Omron Sysmac Studio project RingBufferExample_FallbackLogger (Sysmac Studio 1.62.0.9, StandardProject)
(* Examples for RingBufferLib. *)

# Controller Example: NX102-9000 version 1.64
Task Main (priority 4, period or condition 2000): PseudoMain, ProgramLoader
Task Subsystem (priority 18, period or condition 10000): LogFileWriter, LogSender, RedundantLogSender
Library FileStreamWriterLib 0.0.1 (contents left out)
Library ModeManagerLib 0.0.2 (contents left out)
Library UdpClientLib 0.0.1 (contents left out)
Library RingBufferLib 0.0.2 (contents left out)
Library FileStreamReaderLib 0.0.2 (contents left out)
Library TcpClientLib 0.0.1 (contents left out)

TYPE RetainedRingBufferContext : STRUCT
    Context : stfreakjp\buf\RingBufferContext;
    InitialContext : stfreakjp\buf\RingBufferContext;
    Inited : BOOL;
END_STRUCT END_TYPE

VAR_GLOBAL RETAIN
    gpLoggerBufferContext : RetainedRingBufferContext;
    gpLoggerBuffer : ARRAY[0..32767] OF BYTE;
END_VAR

PROGRAM README
RETURN;
(*

# About This Project
This project demonstrates the RingBufferLib.
It showcases logging by combining RingBufferLib with FileStreamWriterLib, FileStreamReaderLib, and TcpClientLib.
This allows for simultaneous writing of logs to the controller's SD card and sending them to a remote TCP endpoint.

Furthermore, if sending to the TCP endpoint fails, it **falls back** to writing to the SD card.
When the TCP endpoint connection is restored,
the logs that were output during the fallback period are then sent to a dedicated TCP endpoint for fallback logs.

The logger uses its buffer as holding memory to retain values even after a power loss.
Additionally, when writing logs to the SD card or sending them to a remote TCP endpoint,
the output programs also refer to logs the logger wrote before those programs started.

# About the Programs
This project includes the following programs:

* POU/Program/ProgramLoader
    Selects the program to execute.

* POU/Program/PseudoMain
    Continuously generates logs.

* POU/Program/LogFileWriter
    Outputs logs to the controller's SD card.

* POU/Program/LogSender
    Sends logs to a remote TCP endpoint.

* POU/Program/RedundantLogSender
    Sends logs to redundant remote UDP endpoints.

* POU/Program/SimpleTcpMonitor_ps1
    A PowerShell script to set up a TCP endpoint.

* POU/Program/SimpleUdpMonitor_ps1
    A PowerShell script to set up a UDP endpoint.

* POU/Program/StartMultiTcpMonitors_ps1
    A PowerShell script to launch four TCP endpoints in Windows Terminal.

# Usage Steps
Use this program by following these steps:

1.  Configure the project for your environment.
    Match the controller model and ensure access to the network you're using.

2.  Adjust `POU/Program/LogUdpSender` for your environment.
    Change the values of the `REMOTE_ADDR` and `REMOTE_PORT` variables to the remote UDP endpoint that will receive the logs.
	If you're using `POU/Program/RedundantLogUdpSender`, make sure to modify that as well.

3.  Listen for TCP on an appropriate device.
    You can find a reference PowerShell script in `POU/Program/SimpleTcpMonitor_ps1`.
	`StartMultiTcpMonitors_ps1` is a PowerShell script that uses Windows Terminal to launch four TCP endpoints.

4.  Run the program on the controller.   
    Transfer the program to the controller and start its execution.

5.  Confirm that data is being sent to the opened TCP socket.

6.  Confirm that log files are created on the controller's SD card.


# このプロジェクトについて
このプロジェクトは、RingBufferLibの例示です。
RingBufferLibを使用した、FileStreamWriterLib、FileStreamReaderLibとTcpClientLibを組み合わせたロギングをデモします。
ログのコントローラのSDカードへの書き込みとリモートTCPエンドポイントへの送信を同時に行います。
また、TCPエンドポイントへの送信ができないとき、SDカード出力へフォールバックし、
TCPエンドポイントへの送信が復旧すると、フォールバックしたログをフォールバック専用のTCPエンドポイントに送信します。

ロガーは、バッファを保持メモリとして電源断を越えて値を保持します。
また、ログのSDカードへの書き込みとリモートTCPエンドポイントへの送信は、
それら出力プログラムが起動する以前にロガーが書き込んだログも参照して出力します。

# プログラムについて
このプロジェクトは、以下のプログラムを含みます。

* POU/プログラム/ProgramLoader
  実行するプログラムを選択します。

* POU/プログラム/PseudoMain
  ログを生成し続けます。

* POU/プログラム/LogFileWriter
  コントローラのSDカードにログを出力します。

* POU/プログラム/LogSender
  リモートTCPエンドポイントにログを送信します。

* POU/プログラム/RedundantLogSender
  冗長のリモートUDPエンドポイントにログを送信します。

* POU/プログラム/SimpleTcpMonitor_ps1
  TCPエンドポイントを立ち上げるPowerShellスクリプトです。

* POU/プログラム/SimpleUdpMonitor_ps1
  UDPエンドポイントを立ち上げるPowerShellスクリプトです。

* POU/プログラム/StartMultiTcpMonitors_ps1
  Windows Terminalで4つのTCPエンドポイントを立ち上げるPowerShellスクリプトです。

# 使用手順
このプログラムは、以下の手順で使用します。

1.  プロジェクトの構成を使用環境に合わせる
    コントローラの型式を合わせ、使用するネットワークにアクセスできるようにします。
  
2.  `POU/プログラム/LogSender`を使用環境に合わせる
    `REMOTE_ADDR`と`REMOTE_PORT`変数の値をログを受信するリモートTCPエンドポイントに変更します。
	`POU/プログラム/RedundantLogSender`を使用する場合、そちらも変更します。
  
3.  適当な端末でTCPをリッスンする
    `POU/プログラム/SimpleTcpMonitor_ps1`に参考のPowerShellスクリプトがあります。
	`StartMultiTcpMonitors_ps1`は、Windows Terminalを使用して4つのTCPエンドポイントを立ち上げるPowerShellスクリプトです。

4.  コントローラでプログラムを動作させる
    プログラムをコントローラに転送して動作させます。
  
5.  待ち受けているTCPソケットにデータが送られてくることを確認する

6.  コントローラのSDカードにログファイルが作成されていることを確認する


For the parts to which I have rights, I follow POU/Program/LICENSE.
You are free to use and modify it, but we are not responsible for any damage or loss related to it.

(c) 2025 KITA Munemitsu

*)
END_PROGRAM

PROGRAM ProgramLoader
VAR
    iModeManager : ModeManagerContext;
    RUN_MODE : STRING[128];
END_VAR
(*

# About This Program
This program is the selector for the execution program.
Specify the operation mode with "RUN_MODE" in "Configuration".


# このプログラムについて
このプログラムは、実行プログラムのセレクタです。
"Configuration"の"RUN_MODE"で動作モードを指定します。


(c) 2025 KITA Munemitsu

*)

// Configuration
IF P_First_Run THEN
	// "run:standalone", "run" or "run:redundant".
	RUN_MODE := 'run';
END_IF;

IF P_First_Run THEN
	ModeManager_init(Context:=iModeManager,
					 Name:='ProgramLoader',
					 OnSuccessStop:=TRUE,
					 OnFailStop:=FALSE,
					 OnFailAlarm:=TRUE,
					 AlarmCode:=1);

	ModeSet(Context:=iModeManager);
		// Logs are output to the controller's SD card.
		Mode(Context:=iModeManager, Name:='run:standalone');
			ModeUnit(Context:=iModeManager, Name:='PseudoMain');
			ModeUnit(Context:=iModeManager, Name:='LogFileWriter');

		// It outputs logs to the controller's SD card and to a remote TCP endpoint.
		Mode(Context:=iModeManager, Name:='run');
			ModeUnit(Context:=iModeManager, Name:='PseudoMain');
			ModeUnit(Context:=iModeManager, Name:='LogFileWriter');
			ModeUnit(Context:=iModeManager, Name:='LogSender');

		// It outputs logs to the controller's SD card and to two remote TCP endpoints.
		Mode(Context:=iModeManager, Name:='run:redundant');
			ModeUnit(Context:=iModeManager, Name:='PseudoMain');
			ModeUnit(Context:=iModeManager, Name:='LogFileWriter');
			ModeUnit(Context:=iModeManager, Name:='LogSender');
			ModeUnit(Context:=iModeManager, Name:='RedundantLogSender');
	ModeSetClose(Context:=iModeManager);
	
	ModeManager_selectMode(Context:=iModeManager, Name:=RUN_MODE);
END_IF;

ModeManager_activate(Context:=iModeManager);
END_PROGRAM

PROGRAM PseudoMain
VAR
    LOGGING_INTERVAL : UINT;
END_VAR
VAR RETAIN
    iCounter : ULINT := 0;
END_VAR
VAR
    iMsg : STRING[1024];
    iWaitTick : UINT;
END_VAR
VAR RETAIN
    iForceClear : BOOL;
END_VAR
VAR_EXTERNAL
    gpLoggerBuffer : ARRAY[0..32767] OF BYTE;
    gpLoggerBufferContext : RetainedRingBufferContext;
END_VAR
(*

# About This Program
This program will keep writing logs.
Setting `iForceClear` to "TRUE" will force initialization.


# このプログラムについて
このプログラムは、ログを書き続けます。
`iForceClear`を"TRUE"にすることで、強制的に初期化します。


(c) 2025 KITA Munemitsu

*)

// Configuration
IF P_First_Run THEN
	LOGGING_INTERVAL := 1;
	// iForceClear := FALSE;
END_IF;

IF P_First_Run THEN
	// Setup Logger.
	RetainedLogger_init(Context:=gpLoggerBufferContext,
						Buffer:=gpLoggerBuffer,
						ForceClear:=iForceClear);
	IF iForceClear THEN
		iCounter := 0;
		iForceClear := FALSE;
	END_IF;
	
	iMsg := CONCAT('{"boot":true',
				   CONCAT(',"lastcount":', ULINT_TO_STRING(iCounter)),
				   CONCAT(',"timestamp":"', DtToString(GetTime()), '"'),
				   '}$L');
	RetainedLogger_write(Context:=gpLoggerBufferContext,
						 Buffer:=gpLoggerBuffer,
						 Message:=iMsg);
	
	iWaitTick := LOGGING_INTERVAL;
END_IF;

// Logging at regular intervals.
Dec(iWaitTick);
IF iWaitTick < 1 THEN
	Inc(iCounter);
	iMsg := CONCAT('{"counter":', ULINT_TO_STRING(iCounter),
				   ',"timestamp":"', DtToString(GetTime()),
				   '"}$L');
	RetainedLogger_write(Context:=gpLoggerBufferContext,
						 Buffer:=gpLoggerBuffer,
						 Message:=iMsg);
	
	iWaitTick := LOGGING_INTERVAL;
END_IF;
END_PROGRAM

PROGRAM LogFileWriter
VAR
    LOG_PATH : STRING[64];
    iLogFileWriter : stfreakjp\fileio\FileStreamWriter;
    iLogFileWriterContext : stfreakjp\fileio\FileStreamWriterContext;
    iLogFileWriterBufferContext : stfreakjp\buf\RingBufferContext;
    iLogFileWriterBuffer : ARRAY[0..65534] OF BYTE;
END_VAR
VAR RETAIN
    ipLoggerWrittenTracker : stfreakjp\buf\RingBufferContext;
END_VAR
VAR_EXTERNAL
    gpLoggerBuffer : ARRAY[0..32767] OF BYTE;
    gpLoggerBufferContext : RetainedRingBufferContext;
END_VAR
(*

# About This Program
This program keeps track of the logger's buffer writes and outputs them to a file.


# このプログラムについて
このプログラムは、ロガーのバッファ書き込みを追跡してファイルに出力し続けます。


(c) 2025 KITA Munemitsu

*)

// Configuration
IF P_First_Run THEN
	LOG_PATH := '/log.txt';
END_IF;

IF P_First_Run THEN
	// Setup Log writer.
	RingBuffer_init(Context:=iLogFileWriterBufferContext,
					Buffer:=iLogFileWriterBuffer);	
	FileStreamWriter_configure(Context:=iLogFileWriterContext,
							   Activate:=TRUE,
							   Path:=LOG_PATH,
							   FileOpenMode:=_eFOPEN_MODE#_WRITE_APPEND,
							   FlushThreshold:=(SizeOfAry(iLogFileWriterBuffer) / 2),
							   FlushOnDeactivate:=TRUE);
	iLogFileWriter.Enable := TRUE;
	
	// Tracks Logger writes.
	RetainedRingBuffer_createWriteTracker(
		Target:=gpLoggerBufferContext,
		Tracker:=ipLoggerWrittenTracker);
END_IF;

// Gets the difference of the logger buffer into the log writer's write buffer.
RetainedRingBuffer_pullWrite(Context:=iLogFileWriterBufferContext,
							 Buffer:=iLogFileWriterBuffer,
							 Tracker:=ipLoggerWrittenTracker,
							 Tracked:=gpLoggerBufferContext,
							 TrackedBuffer:=gpLoggerBuffer);
iLogFileWriter(Context:=iLogFileWriterContext,
			   BufferContext:=iLogFileWriterBufferContext,
			   Buffer:=iLogFileWriterBuffer);
END_PROGRAM

PROGRAM LogSender
VAR CONSTANT
    LOG_SENDER_RESET_PAYLOAD : STRING[8] := '$$R$$L$$R$$L';
END_VAR
VAR
    FALLBACK_FILE_PATH : STRING[64];
    REMOTE_ADDR : STRING[256];
    REMOTE_PORT : UINT;
    REMOTE_FALLBACK_PORT : UINT;
    WAIT_TICKS_UNTILE_STABLE : UINT;
END_VAR
VAR CONSTANT
    STATE_REMOTE_ACTIVE : UINT := 0;
    STATE_REMOTE_INACTIVE : UINT := 1;
    STATE_FALLBACK_WAIT : UINT := 10;
    STATE_FALLBACK_HALT : UINT := 5;
    STATE_FALLBACK_ACTIVE : UINT := 20;
    STATE_FALLBACK_SENDER_ERROR : UINT := 900;
    STATE_FALLBACK_SENDER_INACTIVE : UINT := 0;
    STATE_FALLBACK_SENDER_HALT : UINT := 5;
    STATE_FALLBACK_SENDER_ACTIVE : UINT := 20;
END_VAR
VAR
    iLogSenderClient : stfreakjp\net\TcpSendClient;
    iLogSenderContext : stfreakjp\net\TcpClientContext;
END_VAR
VAR RETAIN
    iLogSenderBufferContext : stfreakjp\buf\RingBufferContext;
    iLogSenderBuffer : ARRAY[0..65534] OF BYTE;
    ipLoggerWrittenTracker : stfreakjp\buf\RingBufferContext;
END_VAR
VAR
    iFallbackLogWriter : stfreakjp\fileio\FileStreamWriter;
    iFallbackLogWriterContext : stfreakjp\fileio\FileStreamWriterContext;
END_VAR
VAR RETAIN
    iFallbackLogBufferContext : stfreakjp\buf\RingBufferContext;
    iFallbackLogBuffer : ARRAY[0..32767] OF BYTE;
END_VAR
VAR
    iFallbackLogReader : stfreakjp\fileio\FileStreamReader;
    iFallbackLogReaderContext : stfreakjp\fileio\FileStreamReaderContext;
    iFallbackLogReaderBufferContext : stfreakjp\buf\RingBufferContext;
    iFallbackLogReaderBuffer : ARRAY[0..8191] OF BYTE;
    iFallbackLogSenderContext : stfreakjp\net\TcpClientContext;
    iFallbackLogSender : stfreakjp\net\TcpSendClient;
    iState : UINT := 0;
    iStateFallback : UINT := 0;
    iStateFallbackSender : UINT := 0;
    iWaitTick : UINT;
    iFileOpenMode : _eFOPEN_MODE;
    iErrorID : WORD;
END_VAR
VAR_EXTERNAL
    gpLoggerBufferContext : RetainedRingBufferContext;
    gpLoggerBuffer : ARRAY[0..32767] OF BYTE;
END_VAR
(*

# About This Program
This program continuously **tracks logger buffer writes and sends them to a remote TCP endpoint.
If sending to the TCP endpoint isn't possible, it falls back to outputting to an SD card.
Once the TCP endpoint connection is restored,
the logs written to the SD card are then sent to a dedicated remote TCP endpoint for fallback logs.

Before running it, you must change the "REMOTE_ADDR" in "Configuration" to adjust your environment.

## Regarding Failures During Fallback
Failures can occur even while in fallback mode.
Here's how they impact the system.

*   Power Loss During Fallback Output
    Since the fallback buffer is retained, the system will output the file upon power-up.
 
*   Writer Error During Fallback Output
    Data loss is expected as autonomous recovery isn't feasible.
	The fallback functionality will cease operation.
	
*   Buffer Overflow Before Fallback Output Starts
    This will result in data loss.

*   Fallback Occurs While Sending Fallback Logs
    The system will **append new output to the existing file.
	
*   Power Loss During Fallback Transmission
    All data will be **re-sent upon power-up**.

*   Reader Error During Fallback Transmission
    If the file doesn't exist, there will be data loss.
	Fallback transmission will stop.

*   Sender Error During Fallback Transmission
    Retries will occur as long as the main sender is operational.
	If the main sender is down, fallback transmission will stop.


# このプログラムについて
このプログラムは、ロガーのバッファ書き込みを追跡してリモートのTCPエンドポイントに送信し続けます。
また、TCPエンドポイントへの送信ができないときはフォールバックしてSDカードに出力します。
そして、TCPエンドポイントへの送信が可能になるとSDカードに書き出したログを、
フォールバックを専用に受信するリモートのTCPエンドポイントに送信します。
実行前に"Configuration"の"REMOTE_ADDR"を使用環境に合わせる必要があります。

## フォールバック中の障害について
フォールバック中にも障害が発生する可能性があります。
フォールバック中の障害の影響は、以下です。

*   フォールバック出力中に電源断
    フォールバックバッファが保持なので電源入時にファイル出力。

*   フォールバック出力中にWriterがエラー
    自律的な回復が見込めないのでデータ喪失。
    フォールバック機能停止。

*   フォールバック出力開始までにバッファがオーバーフロー
    データ喪失。

*   フォールバック送信中にフォールバック発生
    ファイルに追記で出力。
  
*   フォールバック送信中に電源断
    電源入時に全て再送信。

*   フォールバック送信中にReaderがエラー
    ファイルが存在しなければデータ喪失。
    フォールバック送信停止。
  
*   フォールバック送信中にSenderがエラー
    主Senderが落ちない限り再試行。
    主Senderが落ちているときフォールバック送信停止。


(c) 2025 KITA Munemitsu

*)

// Configuration.
IF P_First_Run THEN
	REMOTE_ADDR := 'YOUR_REMOTE_DEVICE';
	REMOTE_PORT := 12101;
	REMOTE_FALLBACK_PORT := 12102;
	FALLBACK_FILE_PATH := '/log_fallback.txt';
	WAIT_TICKS_UNTILE_STABLE := 1000;
END_IF;

IF P_First_Run THEN	
	// Setup Log sender.
	//
	// The log sender monitors the logger buffer and sends the written logs.
	IF NOT RingBuffer_isInitialized(Context:=iLogSenderBufferContext) THEN
		RingBuffer_init(Context:=iLogSenderBufferContext,
						Buffer:=iLogSenderBuffer);
	END_IF;
	TcpClient_configure(Context:=iLogSenderContext,
						Activate:=TRUE,
						Destination:=REMOTE_ADDR,
						DestinationPort:=REMOTE_PORT,
						Port:=0,
						UseSend:=TRUE,
						ConnectRetryTimes:=360,
						ConnectRetryInterval:=50,
						ConnectTimeout:=10);
	iLogSenderClient.Enable := TRUE;
	
	// Tracks logger writes.
	RetainedRingBuffer_createWriteTracker(Target:=gpLoggerBufferContext,
										  Tracker:=ipLoggerWrittenTracker);

	// Sends the log sender reset payload first.
	RingBuffer_writeString(Context:=iLogSenderBufferContext,
						   Buffer:=iLogSenderBuffer,
						   Value:=LOG_SENDER_RESET_PAYLOAD);
END_IF;

// Log sender task.
CASE iState OF
	// STATE_REMOTE_ACTIVE
	0:		
		IF TcpClient_isReconnecting(Context:=iLogSenderContext) THEN
			RingBuffer_transferFully(Source:=iLogSenderBufferContext,
									 SourceBuffer:=iLogSenderBuffer,
									 Destination:=iFallbackLogBufferContext,
									 DestinationBuffer:=iFallbackLogBuffer);
			
			iState := STATE_REMOTE_INACTIVE;
		ELSE
			RetainedRingBuffer_pullWrite(Context:=iLogSenderBufferContext,
										 Buffer:=iLogSenderBuffer,
										 Tracker:=ipLoggerWrittenTracker,
										 Tracked:=gpLoggerBufferContext,
										 TrackedBuffer:=gpLoggerBuffer);
		END_IF;
		
	// STATE_REMOTE_INACTIVE
	1:	
		IF TcpClient_isActive(Context:=iLogSenderContext) THEN			
			iState := STATE_REMOTE_ACTIVE;
		ELSE
			RetainedRingBuffer_pullWrite(Context:=iFallbackLogBufferContext,
										 Buffer:=iFallbackLogBuffer,
										 Tracker:=ipLoggerWrittenTracker,
										 Tracked:=gpLoggerBufferContext,
										 TrackedBuffer:=gpLoggerBuffer);
			IF NOT TcpClient_isReconnecting(Context:=iLogSenderContext) THEN
				Inc(iState);
			END_IF;
		END_IF;

	// STATE_DOWN
	2:
		RetainedRingBuffer_pullWrite(Context:=iFallbackLogBufferContext,
									 Buffer:=iFallbackLogBuffer,
									 Tracker:=ipLoggerWrittenTracker,
									 Tracked:=gpLoggerBufferContext,
									 TrackedBuffer:=gpLoggerBuffer);			
END_CASE;
iLogSenderClient(Context:=iLogSenderContext,
				 SendBufferContext:=iLogSenderBufferContext,
				 SendBuffer:=iLogSenderBuffer);

// Fallback file writer task.
CASE iStateFallback OF
	// STATE_FALLBACK_INIT
	0:
		IF RingBuffer_isReadable(Context:=iFallbackLogBufferContext) THEN
			iStateFallback := STATE_FALLBACK_ACTIVE;
		ELSE
			RingBuffer_init(Context:=iFallbackLogBufferContext,
							Buffer:=iFallbackLogBuffer);
			
			iStateFallback := STATE_FALLBACK_WAIT;
		END_IF;
	
	// STATE_FALLBACK_HALT
	// 5:
		
	// STATE_FALLBACK_WAIT
	10:
		CASE iState OF
			// STATE_INACTIVE
			1: iStateFallback := STATE_FALLBACK_ACTIVE;
		END_CASE;
	
	// STATE_FALLBACK_ACTIVE
	20:
		CASE iStateFallbackSender OF
			// STATE_FALLBACK_SENDER_INACTIVE
			0: iFileOpenMode := _eFOPEN_MODE#_WRITE_CREATE;
		ELSE
			iFileOpenMode := _eFOPEN_MODE#_WRITE_APPEND;
		END_CASE;
		FileStreamWriter_configure(Context:=iFallbackLogWriterContext,
								   Activate:=TRUE,
								   Path:=FALLBACK_FILE_PATH,
								   FileOpenMode:=iFileOpenMode,
								   FlushThreshold:=(SizeOfAry(iFallbackLogBuffer) / 2),
								   FlushOnDeactivate:=TRUE);
		iFallbackLogWriter.Enable := TRUE;
		
		Inc(iStateFallback);
	21:
		CASE iState OF
			// STATE_REMOTE_ACTIVE
			0:
				FileStreamWriter_deactivate(Context:=iFallbackLogWriterContext);
				iFallbackLogWriter.Enable := FALSE;

				Inc(iStateFallback);
		ELSE			
			IF FileStreamWriter_hasError(Context:=iFallbackLogWriterContext) THEN
				FileStreamWriter_deactivate(Context:=iFallbackLogWriterContext);
				iFallbackLogWriter.Enable := FALSE;
				
				iStateFallback := STATE_FALLBACK_HALT;
			ELSE
				RetainedRingBuffer_pullWrite(Context:=iFallbackLogBufferContext,
											 Buffer:=iFallbackLogBuffer,
											 Tracker:=ipLoggerWrittenTracker,
											 Tracked:=gpLoggerBufferContext,
											 TrackedBuffer:=gpLoggerBuffer);	
			END_IF;
		END_CASE;
	22:
		IF NOT iFallbackLogWriter.Busy THEN
			IF FileStreamWriter_hasError(COntext:=iFallbackLogWriterContext) THEN
				iStateFallback := STATE_FALLBACK_HALT;
			ELSE	
				iWaitTick := MAX(UINT#1, WAIT_TICKS_UNTILE_STABLE);
			
				Inc(iStateFallback);
			END_IF;
		END_IF;
	23:
		Dec(iWaitTick);
		CASE iState OF
			// STATE_REMOTE_INACTIVE
			1:
				FileStreamWriter_configure(Context:=iFallbackLogWriterContext,
										   Activate:=TRUE,
										   Path:=FALLBACK_FILE_PATH,
										   FileOpenMode:=_eFOPEN_MODE#_WRITE_APPEND,
										   FlushThreshold:=(SizeOfAry(iFallbackLogBuffer) / 2),
										   FlushOnDeactivate:=TRUE);
				iFallbackLogWriter.Enable := TRUE;

				iStateFallback := iStateFallback - 2;
		ELSE
			IF iWaitTick < 1 THEN
				CASE iStateFallbackSender OF
					// STATE_FALLBACK_SENDER_INACTIVE
					0: iStateFallbackSender := STATE_FALLBACK_SENDER_ACTIVE;
				END_CASE;
				
				iStateFallback := STATE_FALLBACK_WAIT;
			END_IF;
		END_CASE;
END_CASE;
iFallbackLogWriter(Context:=iFallbackLogWriterContext,
				   BufferContext:=iFallbackLogBufferContext,
				   Buffer:=iFallbackLogBuffer);

// Fallbacked log sender task.
CASE iStateFallbackSender OF
	// STATE_FALLBACK_SENDER_INACTIVE
	// 0:
	
	// STATE_FALLBACK_SENDER_HALT
	// 5:
	
	// STATE_FALLBACK_SENDER_ACTIVE
	20:
		RingBuffer_init(Context:=iFallbackLogReaderBufferContext,
						Buffer:=iFallbackLogReaderBuffer);
		TcpClient_configure(Context:=iFallbackLogSenderContext,
							Activate:=TRUE,
							Destination:=REMOTE_ADDR,
							DestinationPort:=REMOTE_FALLBACK_PORT,
							Port:=0,
							UseSend:=TRUE,
							ConnectRetryTimes:=20,
							ConnectRetryInterval:=100,
							ConnectTimeout:=100);
		iFallbackLogSender.Enable := TRUE;
		FileStreamReader_configure(Context:=iFallbackLogReaderContext,
								   Activate:=TRUE,
								   Path:=FALLBACK_FILE_PATH,
								   ReadThreshold:=(SizeOfAry(iFallbackLogReaderBuffer) / 2));
		iFallbackLogReader.Enable := TRUE;
		
		Inc(iStateFallbackSender);
	21:
		IF TcpClient_hasError(Context:=iFallbackLogSenderContext) THEN
			iStateFallbackSender := iStateFallbackSender + 6;
		ELSIF TcpClient_isActive(Context:=iFallbackLogSenderContext) THEN
			FileStreamReader_activate(Context:=iFallbackLogReaderContext);
			
			Inc(iStateFallbackSender);
		END_IF;
	22:
		IF TcpClient_hasError(Context:=iFallbackLogSenderContext)
			OR FileStreamReader_hasError(Context:=iFallbackLogReaderContext)
		THEN
			iStateFallbackSender := iStateFallbackSender + 5;
		ELSIF FileStreamReader_isEOF(Context:=iFallbackLogReaderContext) THEN			
			Inc(iStateFallbackSender);
		END_IF;
	23:
		IF TcpClient_hasError(Context:=iFallbackLogSenderContext) THEN
			iStateFallbackSender := iStateFallbackSender + 4;
		ELSIF NOT RingBuffer_isReadable(Context:=iFallbackLogReaderBufferContext) THEN
			iStateFallbackSender := iStateFallbackSender + 4;
		END_IF;
	27:
		TcpClient_deactivate(Context:=iFallbackLogSenderContext);
		FileStreamReader_deactivate(Context:=iFallbackLogReaderContext);
		iFallbackLogSender.Enable := FALSE;
		iFallbackLogReader.Enable := FALSE;
		
		Inc(iStateFallbackSender);
	28:
		IF NOT (iFallbackLogReader.Busy OR iFallbackLogReader.Busy) THEN
			Inc(iStateFallbackSender);
		END_IF;
	29:
		IF TcpClient_hasError(Context:=iFallbackLogSenderContext)
			OR FileStreamReader_getError(Context:=iFallbackLogReaderContext, ErrorID=>iErrorID)
		THEN
			CASE WORD_TO_UINT(iErrorID) OF
				16#0000, // None.
				16#1405, // Accessing file.
				16#140B: // Exceeding maximum number of open files.
					iStateFallbackSender := STATE_FALLBACK_SENDER_ERROR;
			ELSE
				iStateFallbackSender := STATE_FALLBACK_SENDER_HALT;
			END_CASE;
		ELSE
			iStateFallbackSender := STATE_FALLBACK_SENDER_INACTIVE;
		END_IF;
	
	// STATE_FALLBACK_SENDER_ERROR
	900:
		CASE iState OF
			// STATE_ACTIVE
			0: iStateFallbackSender := STATE_FALLBACK_SENDER_ACTIVE;
			// STATE_DOWN
			2: iStateFallbackSender := STATE_FALLBACK_SENDER_HALT;
		END_CASE;
END_CASE;
iFallbackLogReader(Context:=iFallbackLogReaderContext,
				   BufferContext:=iFallbackLogReaderBufferContext,
				   Buffer:=iFallbackLogReaderBuffer);
iFallbackLogSender(Context:=iFallbackLogSenderContext,
				   SendBufferContext:=iFallbackLogReaderBufferContext,
				   SendBuffer:=iFallbackLogReaderBuffer);
END_PROGRAM

PROGRAM RedundantLogSender
VAR CONSTANT
    LOG_SENDER_RESET_PAYLOAD : STRING[8] := '$$R$$L$$R$$L';
END_VAR
VAR
    REMOTE_ADDR : STRING[256];
    REMOTE_PORT : UINT;
    SENDER_PORT : UINT;
    iLogSenderUdpClient : stfreakjp\net\UdpSendClient;
    iLogSenderContext : stfreakjp\net\UdpClientContext;
    iLogSenderSendBufferContext : stfreakjp\buf\RingBufferContext;
    iLogSenderSendBuffer : ARRAY[0..8191] OF BYTE;
END_VAR
VAR RETAIN
    ipLoggerWrittenTracker : stfreakjp\buf\RingBufferContext;
END_VAR
VAR_EXTERNAL
    gpLoggerBufferContext : RetainedRingBufferContext;
    gpLoggerBuffer : ARRAY[0..32767] OF BYTE;
END_VAR
(*

# About This Program
This program acts as a redundancy for log transmission.
Before running it, you must change the "REMOTE_ADDR" in "Configuration" to adjust your environment.


# このプログラムについて
このプログラムは、ログ送信の冗長機能として動作します。
実行前に"Configuration"の"REMOTE_ADDR"を使用環境に合わせる必要があります。


(c) 2025 KITA Munemitsu

*)

// Configuration.
IF P_First_Run THEN
	REMOTE_ADDR := 'YOUR_REMOTE_DEVICE';
	REMOTE_PORT := 12002;
	SENDER_PORT := 12002;
END_IF;

IF P_First_Run THEN	
	// Setup Log sender.
	//
	// The log sender monitors the logger buffer and sends the written logs.
	//
	RingBuffer_init(Context:=iLogSenderSendBufferContext,
					Buffer:=iLogSenderSendBuffer);
	UdpClient_configure(Context:=iLogSenderContext,
						Activate:=TRUE,
						Destination:=REMOTE_ADDR,
						DestinationPort:=REMOTE_PORT,
						Port:=SENDER_PORT,
						UseSend:=TRUE);
	iLogSenderUdpClient.Enable := TRUE;
	
	// Tracks logger writes.
	RetainedRingBuffer_createWriteTracker(
		Target:=gpLoggerBufferContext,
		Tracker:=ipLoggerWrittenTracker);

	// Sends the log sender reset payload first.
	RingBuffer_writeString(Context:=iLogSenderSendBufferContext,
						   Buffer:=iLogSenderSendBuffer,
						   Value:=LOG_SENDER_RESET_PAYLOAD);
END_IF;

// Gets the difference of the logger buffer into the log sender's sending buffer.
RetainedRingBuffer_pullWrite(Context:=iLogSenderSendBufferContext,
							 Buffer:=iLogSenderSendBuffer,
							 Tracker:=ipLoggerWrittenTracker,
							 Tracked:=gpLoggerBufferContext,
							 TrackedBuffer:=gpLoggerBuffer);
iLogSenderUdpClient(Context:=iLogSenderContext,
					SendBufferContext:=iLogSenderSendBufferContext,
					SendBuffer:=iLogSenderSendBuffer);
END_PROGRAM

PROGRAM SimpleTcpMonitor_ps1
RETURN;
(*

Below is a PowerShell script that opens and listens on a TCP socket.


以下は、TCPソケットをオープンして待ち受けるPowerShellスクリプトです。

```powershell:simple-tcp-monitor.ps1
param(
    [Parameter(Mandatory=$false, Position=0)][int]$Port = 12101,
    [Parameter(Mandatory=$false, Position=0)][int]$ReadInterval = 50,
    [Parameter(Mandatory=$false, Position=1)][string]$Mode = 'jsonl'
)

function Mode-Jsonl {
    param(
        [int]$Port,
        [int]$ReadInterval
    )
    $listenerEndPoint = New-Object IPEndpoint([System.Net.IPAddress]::Any, $Port)
    $tcpListener = New-Object System.Net.Sockets.TCPListener($listenerEndpoint)
    $client = $null
    $clientStream = $null
    $reader = $null
    $task = $null
    $entity = $null
    $prevEntity = $null

    try {
        $tcpListener.Start()
        while ($true) {
            # Wait for client connection.
            if ($null -eq $client) {
                if ($null -eq $task) {
                    $task = $tcpListener.AccepttcpClientAsync()
                }
                if (-not $task.Wait(200)) {
                    continue
                }

                $client = $task.GetAwaiter().GetResult();
                $clientStream = $client.GetStream()
                $reader = New-Object System.IO.StreamReader($clientStream)
                $task = $null
            }
            if ($reader.EndOfStream) {
                $reader.Close()
                $clientStream.Close()
                $client.Close()
                $task = $null
                $reader = $null
                $clientStream = $null
                $client = $null
                $entity = $null
                $prevEntity = $null
                continue
            }

            # Waiting to receive data.
            try {
                if ($null -eq $task) {
                    $task = $reader.ReadLineAsync()
                }

                if (-not $task.Wait($ReadInterval)) {
                    continue
                }
                $entity = $task.GetAwaiter().GetResult();
                $task = $null
            }
            catch {
                Write-Host "error: $($_.Exception.Message)"
                $reader.Close()
                $clientStream.Close()
                $client.Close()
                $reader = $null
                $ClientStream = $null
                $client = $null
            }

            if ($null -ne $entity) {
                if ("" -eq $entity) {
                    if ("" -eq $prevEntity) {
                        Write-Host 'reset'
                    }
                } else {
                    try {
                        $entity | ConvertFrom-Json | Write-Host
                    }
                    catch {
                        Write-Host "error payload: ${entity}"
                    }
                }
            }

            $prevEntity = $entity
            $entity = $null
        }
    }
    catch {
        Write-Host "error: $($_.Exception.Message)"
    }
    finally {
        if ($client) {
            $reader.Close()
            $clientStream.Close()
            $client.Close()
        }
        $tcpListener.Stop()
    }
}

function Mode-Raw {
    param(
        [string]$Port,
        [int]$ReadInterval
    )
    $listenerEndPoint = New-Object IPEndpoint([System.Net.IPAddress]::Any, $Port)
    $tcpListener = New-Object System.Net.Sockets.TCPListener($listenerEndpoint)
    $client = $null
    $clientStream = $null
    $reader = $null
    $task = $null
    $prevEntity = $null

    try {
        $tcpListener.Start()
        while ($true) {
            # Wait for client connection.
            if ($null -eq $client) {
                if ($null -eq $task) {
                    $task = $tcpListener.AcceptTcpClientAsync()
                }
                if (-not $task.Wait(200)) {
                    continue
                }

                $client = $task.GetAwaiter().GetResult();
                $clientStream = $client.GetStream()
                $reader = New-Object System.IO.StreamReader($clientStream)
                $task = $null
            }
            if ($reader.EndOfStream) {
                $reader.Close()
                $clientStream.Close()
                $client.Close()
                $task = $null
                $reader = $null
                $clientStream = $null
                $client = $null
                $entity = $null
                $prevEntity = $null
                continue
            }

            # Waiting to receive data.
            try {
                if ($null -eq $task) {
                    $task = $reader.ReadLineAsync()
                }

                if (-not $task.Wait($ReadInterval)) {
                    continue
                }
                $entity = $task.GetAwaiter().GetResult();
                $task = $null
            }
            catch {
                Write-Host "error: $($_.Exception.Message)"
                $reader.Close()
                $clientStream.Close()
                $client.Close()
                $reader = $null
                $ClientStream = $null
                $client = $null
            }

            if ($null -ne $entity) {
                if ("" -eq $entity) {
                    if ("" -eq $prevEntity) {
                        Write-Host 'reset'
                    }
                } else {
                    $entity | Write-Host
                }
            }

            $prevEntity = $entity
            $entity = $null
        }
    }
    catch {
        Write-Host "error: $($_.Exception.Message)"
    }
    finally {
        if ($client) {
            $reader.Close()
            $clientStream.Close()
            $client.Close()
        }
        $tcpListener.Stop()
    }
}

switch ( $Mode )
{
    Jsonl { Mode-Jsonl -Port $Port -ReadInterval $ReadInterval }
    Raw   { Mode-Raw -Port $Port -ReadInterval $ReadInterval }
}
```
*)
END_PROGRAM

PROGRAM SimpleUdpMonitor_ps1
RETURN;
(*

Below is a PowerShell script that opens and listens on a UDP socket.


以下は、UDPソケットをオープンして待ち受けるPowerShellスクリプトです。

```powershell:simple-udp-monitor.ps1
param(
    [Parameter(Mandatory=$false, Position=0)][int]$Port = 12001,
    [Parameter(Mandatory=$false, Position=1)][string]$Mode = 'raw'
)

function Mode-Jsonl {
    param(
        [string]$Port
    )

    $udpClient = New-Object System.Net.Sockets.UdpClient($Port)
    try {
        $task = $null
        $RESET_PAYLOAD = "`r`n`r`n"
        $ENTITY_DELIMITER = "`n"
        $ENTITY_MAX_LENGTH = 8192
        $recv = $null
        $payload = $null
        $restPaylod = $null
        $entities = $null
        while ($true) {
            if ($null -eq $task) {
                $task = $udpClient.ReceiveAsync()
            }
            if (-not $task.Wait(20)) {
                continue
            }
            $receiveBytes = $task.GetAwaiter().GetResult();

            $recv = [Text.Encoding]::UTF8.GetString($receiveBytes.Buffer)
            $payload = $recv -split $RESET_PAYLOAD
            if ($payload.length -gt 1) {
                Write-Host 'reset'
                $restPaylod = ""
            }
            $entities = ($restPaylod + $payload[-1]) -split $ENTITY_DELIMITER
                | Where-Object {($_ -ne "") -and ($_.Length -le $ENTITY_MAX_LENGTH)}
            $restPaylod = ""
            foreach ($entity in $entities) {
                try {
                    $entity | ConvertFrom-Json | Write-Host
                }
                catch {
                    if ($entity -eq $entities[-1]) {
                        $restPaylod = $entity
                    }
                }
            }

            $task = $null
        }
    }
    catch {
        Write-Host "error: $($_.Exception.Message)"
    }
    finally {
        $udpClient.Close()
    }
}

function Mode-Raw {
    param(
        [string]$Port
    )

    $udpClient = New-Object System.Net.Sockets.UdpClient($Port)
    try {
        $task = $null
        $message = ''
        while ($true) {
            if ($null -eq $task) {
                $task = $udpClient.ReceiveAsync()
            }
            if (-not $task.Wait(20)) {
                continue
            }
            $receiveBytes = $task.GetAwaiter().GetResult();
            $message = [Text.Encoding]::UTF8.GetString($receiveBytes.Buffer)
            Write-Host $message -NoNewline

            $task = $null
        }
    }
    catch {
        Write-Host "error: $($_.Exception.Message)"
    }
    finally {
        $udpClient.Close()
    }
}

switch ( $Mode ) {
	Jsonl { Mode-Jsonl -Port $Port }
    Raw   { Mode-Raw -Port $Port }
}
```
*)
END_PROGRAM

PROGRAM StartMultiTcpMonitors_ps1
RETURN;
(*

Below is a PowerShell script that launches four "simple-tcp-monitor.ps" files in Windows Terminal.
Run this script while "simple-tcp-monitor.ps1" is in the same folder.


以下は、Windows Terminalで4つの"simple-tcp-monitor.ps"を立ち上げるPowerShellスクリプトです。
"simple-tcp-monitor.ps1"が同じフォルダにある状態で実行します。

```powershell:start-multi-tcp-monitors.ps1
param(
    [Parameter(Mandatory=$false, Position=0)][int[]]$Ports = @(12101, 12102, 13101, 13102),
    [Parameter(Mandatory=$false, Position=1)][string]$Mode = 'jsonl'
)

$scriptFile = "simple-tcp-monitor.ps1"
$scriptDir = Split-Path -Parent $MyInvocation.MyCommand.Definition
$scriptPath = Join-Path $scriptDir $scriptFile
if (-not (Test-Path $scriptPath)) {
    Write-Error "error: Not fount '${scriptFile}' in '${scriptPath}'"
    exit 1
}

$wtCommandString = "pwsh.exe -NoExit -Command ""&{ & `"${scriptPath}`" -Port $($Ports[0]) -Mode `"${Mode}`" }"" ; " + `
                   "split-pane -H pwsh.exe -NoExit -Command ""&{ & `"${scriptPath}`" -Port $($Ports[1]) -Mode `"${Mode}`" }"" ; " + `
                   "split-pane -V pwsh.exe -NoExit -Command ""&{ & `"${scriptPath}`" -Port $($Ports[2]) -Mode `"${Mode}`" }"" ; " + `
                   "split-pane -H pwsh.exe -NoExit -Command ""&{ & `"${scriptPath}`" -Port $($Ports[3]) -Mode `"${Mode}`" }"""

# For debug.
# Write-Host "command: wt.exe $wtCommandString"

Start-Process -FilePath "wt.exe" -ArgumentList $wtCommandString
```
*)
END_PROGRAM

PROGRAM LICENSE
RETURN;
(*
The MIT License (MIT)

Copyright(c) 2025 KITA Munemitsu

Permission is hereby granted, free of charge, to any person obtaining a copy of this software and associated
documentation files (the “Software”), to deal in the Software without restriction, including without limitation
the rights to use, copy, modify, merge, publish, distribute, sublicense, and/or sell copies of the Software,
and to permit persons to whom the Software is furnished to do so, subject to the following conditions:

The above copyright notice and this permission notice shall be included in all copies or substantial portions of the Software.

THE SOFTWARE IS PROVIDED “AS IS”, WITHOUT WARRANTY OF ANY KIND, EXPRESS OR IMPLIED, INCLUDING BUT NOT
LIMITED TO THE WARRANTIES OF MERCHANTABILITY, FITNESS FOR A PARTICULAR PURPOSE AND NONINFRINGEMENT.
IN NO EVENT SHALL THE AUTHORS OR COPYRIGHT HOLDERS BE LIABLE FOR ANY CLAIM, DAMAGES OR OTHER LIABILITY,
WHETHER IN AN ACTION OF CONTRACT, TORT OR OTHERWISE, ARISING FROM, OUT OF OR IN CONNECTION WITH THE SOFTWARE
OR THE USE OR OTHER DEALINGS IN THE SOFTWARE.
*)
END_PROGRAM

FUNCTION RetainedLogger_init : BOOL
VAR_IN_OUT
    Context : RetainedRingBufferContext;
    Buffer : ARRAY[*] OF BYTE;
END_VAR
VAR_INPUT
    ForceClear : BOOL := False;
END_VAR
IF NOT EN THEN
	RetainedLogger_init := FALSE;
	
	RETURN;
END_IF;

RetainedLogger_init
	:= RetainedRingBuffer_init(Context:=Context,
							   Buffer:=Buffer,
							   Force:=ForceClear);
END_FUNCTION

FUNCTION RetainedLogger_write : BOOL
VAR
    iBinMsg : ARRAY[0..4095] OF BYTE;
    iBinMsgSize : UINT;
END_VAR
VAR_IN_OUT
    Context : RetainedRingBufferContext;
    Buffer : ARRAY[*] OF BYTE;
END_VAR
VAR_INPUT
    Message : STRING[1986] := '';
END_VAR
IF NOT EN THEN
	RetainedLogger_write := FALSE;
	
	RETURN;
END_IF;

iBinMsgSize
	:= StringToAry(In:=Message, AryOut:=iBinMsg[0]);
RetainedLogger_write
	:= \\stfreakjp\buf\RingBuffer_write(
						   Context:=Context.Context,
						   Buffer:=Buffer,
						   In:=iBinMsg,
						   Head:=0,
						   Size:=iBinMsgSize,
						   AllowOverWrite:=TRUE);
END_FUNCTION

FUNCTION RetainedRingBuffer_init : BOOL
VAR_IN_OUT
    Context : RetainedRingBufferContext;
    Buffer : ARRAY[*] OF BYTE;
END_VAR
VAR_INPUT
    Force : BOOL := False;
END_VAR
(*

Initializes the RetainedRingBufferContext.


RetainedRingBufferContextを初期化する。


(c) 2025 KITA Munemitsu

*)

IF NOT EN THEN
	RetainedRingBuffer_init := FALSE;
	
	RETURN;
END_IF;

IF NOT Context.Inited OR Force THEN
	\\stfreakjp\buf\RingBuffer_init(
						Context:=Context.Context,
						Buffer:=Buffer);
	Context.Inited := TRUE;
END_IF;

Context.InitialContext := Context.Context;

RetainedRingBuffer_init := TRUE;
END_FUNCTION

FUNCTION RetainedRingBuffer_createWriteTracker : BOOL
VAR_IN_OUT
    Target : RetainedRingBufferContext;
END_VAR
VAR_INPUT
    UseInitial : BOOL := True;
    Force : BOOL := False;
END_VAR
VAR_IN_OUT
    Tracker : stfreakjp\buf\RingBufferContext;
END_VAR
(*

Creates a tracking context for tracking writes to the RetainedRingBuffer.


RetainedRingBufferの書き込みを追跡するための追跡コンテクストを作成する。


(c) 2025 KITA Munemitsu

*)

IF NOT EN
	OR NOT Target.Inited
THEN	
	RetainedRingBuffer_createWriteTracker := FALSE;
	
	RETURN;
END_IF;

// NOTE: Maybe we need a method to determine the validity of a tracker.
IF Target.Context.WriteSize >= Tracker.WriteSize
	AND Tracker.WriteSize <> 0
	AND NOT Force
THEN
	RetainedRingBuffer_createWriteTracker := TRUE;
	
	RETURN;
END_IF;

IF UseInitial THEN
	RetainedRingBuffer_createWriteTracker
		:= \\stfreakjp\buf\RingBuffer_createWriteTracker(
							   Target:=Target.InitialContext,
							   Tracker=>Tracker);
ELSE
	RetainedRingBuffer_createWriteTracker
		:= \\stfreakjp\buf\RingBuffer_createWriteTracker(
							   Target:=Target.Context,
							   Tracker=>Tracker);
END_IF;
END_FUNCTION

FUNCTION RetainedRingBuffer_createReadTracker : BOOL
VAR_IN_OUT
    Target : RetainedRingBufferContext;
END_VAR
VAR_INPUT
    UseInitial : BOOL := True;
    Force : BOOL := False;
END_VAR
VAR_OUTPUT
    Tracker : stfreakjp\buf\RingBufferContext;
END_VAR
(*

Creates a tracking context to track reads of the RetainedRingBuffer.


RetainedRingBufferの読み出しを追跡するための追跡コンテクストを作成する。


(c) 2025 KITA Munemitsu

*)

IF NOT EN
	OR NOT Target.Inited
THEN	
	RetainedRingBuffer_createReadTracker := FALSE;
	
	RETURN;
END_IF;

// NOTE: Maybe we need a method to determine the validity of a tracker.
IF Target.Context.ReadSize >= Tracker.ReadSize
	AND Tracker.ReadSize <> 0
	AND NOT Force
THEN
	RetainedRingBuffer_createReadTracker := TRUE;
	
	RETURN;
END_IF;

IF UseInitial THEN
	RetainedRingBuffer_createReadTracker
		:= \\stfreakjp\buf\RingBuffer_createReadTracker(
							   Target:=Target.InitialContext,
							   Tracker=>Tracker);
ELSE
	RetainedRingBuffer_createReadTracker
		:= \\stfreakjp\buf\RingBuffer_createReadTracker(
							   Target:=Target.Context,
							   Tracker=>Tracker);
END_IF;
END_FUNCTION

FUNCTION RetainedRingBuffer_createTracker : BOOL
VAR_IN_OUT
    Target : RetainedRingBufferContext;
END_VAR
VAR_INPUT
    UseInitial : BOOL := True;
    Force : BOOL := False;
END_VAR
VAR_OUTPUT
    Tracker : stfreakjp\buf\RingBufferContext;
END_VAR
(*

Creates a tracking context for tracking reads and writes to the RetainedRingBuffer.


RetainedRingBufferの読み書きを追跡するための追跡コンテクストを作成する。


(c) 2025 KITA Munemitsu

*)

IF NOT EN THEN	
	RetainedRingBuffer_createTracker := FALSE;
	
	RETURN;
END_IF;

// NOTE: Maybe we need a method to determine the validity of a tracker.
IF Target.Context.WriteSize >= Tracker.WriteSize
	AND Tracker.WriteSize <> 0
	AND Target.Context.ReadSize >= Tracker.ReadSize
	AND Tracker.ReadSize <> 0
	AND NOT Force
THEN
	RetainedRingBuffer_createTracker := TRUE;
	
	RETURN;
END_IF;

IF UseInitial THEN
	RetainedRingBuffer_createTracker
		:= \\stfreakjp\buf\RingBuffer_createTracker(
							   Target:=Target.InitialContext,
							   Tracker=>Tracker);
ELSE
	RetainedRingBuffer_createTracker
		:= \\stfreakjp\buf\RingBuffer_createTracker(
							   Target:=Target.Context,
							   Tracker=>Tracker);
END_IF;
END_FUNCTION

FUNCTION RetainedRingBuffer_pullWrite : BOOL
VAR_IN_OUT
    Context : stfreakjp\buf\RingBufferContext;
    Buffer : ARRAY[*] OF BYTE;
    Tracker : stfreakjp\buf\RingBufferContext;
    Tracked : RetainedRingBufferContext;
    TrackedBuffer : ARRAY[*] OF BYTE;
END_VAR
VAR_INPUT
    AllowOverwrite : BOOL := False;
END_VAR
VAR_OUTPUT
    Missing : BOOL;
    PullSize : UINT;
END_VAR
(*

Gets the write difference from the tracked RetainedRingBuffer.


追跡しているRetainedRingBufferから書き込み差分を取得する。


(c) 2025 KITA Munemitsu

*)

IF NOT EN THEN
	Clear(Missing);
	Clear(PullSize);
	
	RetainedRingBuffer_pullWrite := FALSE;
	
	RETURN;
END_IF;

RetainedRingBuffer_pullWrite
	:= \\stfreakjp\buf\RingBuffer_pullWrite(
						   Context:=Context,
						   Buffer:=Buffer,
						   Tracker:=Tracker,
						   Tracked:=Tracked.Context,
						   TrackedBuffer:=TrackedBuffer,
						   AllowOverwrite:=AllowOverwrite,
						   Missing=>Missing,
						   PullSize=>PullSize);
END_FUNCTION

FUNCTION RetainedRingBuffer_pullRead : BOOL
VAR_IN_OUT
    Context : stfreakjp\buf\RingBufferContext;
    Buffer : ARRAY[*] OF BYTE;
    Tracker : stfreakjp\buf\RingBufferContext;
    Tracked : RetainedRingBufferContext;
    TrackedBuffer : ARRAY[*] OF BYTE;
END_VAR
VAR_INPUT
    AllowOverwrite : BOOL := False;
END_VAR
VAR_OUTPUT
    Missing : BOOL;
    PullSize : UINT;
    Overflow : BOOL;
END_VAR
(*

Gets the read difference from the tracked RetainedRingBuffer.


追跡しているRetainedRingBufferから書き込み差分を取得する。


(c) 2025 KITA Munemitsu

*)

IF NOT EN THEN
	Clear(Missing);
	Clear(PullSize);
	Clear(Overflow);
	
	RetainedRingBuffer_pullRead := FALSE;
	
	RETURN;
END_IF;

RetainedRingBuffer_pullRead
	:= \\stfreakjp\buf\RingBuffer_pullRead(
						   Context:=Context,
						   Buffer:=Buffer,
						   Tracker:=Tracker,
						   Tracked:=Tracked.Context,
						   TrackedBuffer:=TrackedBuffer,
						   AllowOverwrite:=AllowOverwrite,
						   Missing=>Missing,
						   PullSize=>PullSize,
						   Overflow=>Overflow);
END_FUNCTION

FUNCTION RetainedRingBuffer_pull : BOOL
VAR_IN_OUT
    WriteContext : stfreakjp\buf\RingBufferContext;  (* RingBufferContext of the RingBuffer to which the obtained write difference is written. *)
    WriteBuffer : ARRAY[*] OF BYTE;  (* Byte array of the RingBuffer to which the obtained write difference is written. *)
END_VAR
VAR_INPUT
    WriteAllowOverwrite : BOOL := False;  (* Whether to overwrite unread bytes in the RingBuffer where the write difference is written. *)
END_VAR
VAR_IN_OUT
    ReadContext : stfreakjp\buf\RingBufferContext;  (* RingBufferContext of the RingBuffer to which the obtained read difference is written. *)
    ReadBuffer : ARRAY[*] OF BYTE;  (* Byte array of the RingBuffer to which the obtained read difference is written. *)
END_VAR
VAR_INPUT
    ReadAllowOverwrite : BOOL := False;  (* Whether to overwrite unread bytes in the RingBuffer where the read difference is written. *)
END_VAR
VAR_IN_OUT
    Tracker : stfreakjp\buf\RingBufferContext;
    Tracked : RetainedRingBufferContext;
    TrackedBuffer : ARRAY[*] OF BYTE;
END_VAR
VAR_OUTPUT
    WriteMissing : BOOL;
    WritePullSize : UINT;
    ReadMissing : BOOL;
    ReadPullSize : UINT;
    Overflow : BOOL;
END_VAR
(*

Gets the difference from the tracked RetainedRingBuffer.


追跡しているRetainedRingBufferから差分を取得する。

(c) 2025 KITA Munemitsu

*)

IF NOT EN THEN
	Clear(WriteMissing);
	Clear(WritePullSize);
	Clear(ReadMissing);
	Clear(ReadPullSize);
	Clear(Overflow);
	
	RetainedRingBuffer_pull := FALSE;
	
	RETURN;
END_IF;

RetainedRingBuffer_pull
	:= \\stfreakjp\buf\RingBuffer_pull(
						   WriteContext:=WriteContext,
						   WriteBuffer:=WriteBuffer,
						   WriteAllowOverwrite:=WriteAllowOverwrite,
						   ReadContext:=ReadContext,
						   ReadBuffer:=ReadBuffer,
						   ReadAllowOverwrite:=ReadAllowOverwrite,
						   Tracker:=Tracker,
						   Tracked:=Tracked.Context,
						   TrackedBuffer:=TrackedBuffer,
						   WriteMissing=>WriteMissing,
						   WritePullSize=>WritePullSize,
						   ReadMissing=>ReadMissing,
						   ReadPullSize=>ReadPullSize,
						   Overflow=>Overflow);
END_FUNCTION

FUNCTION RingBuffer_writeString : BOOL
VAR
    iBinValue : ARRAY[0..4095] OF BYTE;
    iBinValueSize : UINT;
END_VAR
VAR_IN_OUT
    Context : stfreakjp\buf\RingBufferContext;
    Buffer : ARRAY[*] OF BYTE;
END_VAR
VAR_INPUT
    Value : STRING[1986] := '';
END_VAR
IF NOT EN THEN
	RingBuffer_writeString := FALSE;
	
	RETURN;
END_IF;

iBinValueSize
	:= StringToAry(In:=Value, AryOut:=iBinValue[0]);
RingBuffer_writeString
	:= \\stfreakjp\buf\RingBuffer_write(
						   Context:=Context,
						   Buffer:=Buffer,
						   In:=iBinValue,
						   Head:=0,
						   Size:=iBinValueSize,
						   AllowOverWrite:=TRUE);
END_FUNCTION